(* Schneider Machine Expert - Basic project Temporizador, file version 2.7.0.0 *)
(* ProjectInformations: Name=Nuevo proyecto *)

HARDWARE
  Cpu 0: TM221C24R
  EthernetConfiguration: NetworkName=M221, IpAllocationMode=FixedAddress, IpAddress=0.0.0.0, SubnetMask=0.0.0.0
  SerialLineConfiguration: Baud=Baud19200, Parity=ParityEven, DataBits=DataBits8, StopBits=StopBits1, PhysicalMedium=PhysicalMediumRs485, TransmissionMode=TransmissionModeModbusRtu, SlaveId=1, Addressing=SlaveAddressing
  MastTask: UsePeriodScanMode=false, PeriodScan=100
  FastTask: Period=255
  CpuBehavior: StartingMode=StartAsPreviousState, AutoSaveRamOnEeprom=true, WatchdogPeriod=250

SYMBOLS  (address, symbol, comment, settings)
  %M0         "Fill"
  %M1         "Discharge"
  %M3         "Fill valve"
  %M4         "Fillin"
  %M5         "Discharge valve"
  %M6         "Discharging"
  %TM0        "Timer Fill"  [Type=TP, Preset=10, Base=OneSecond]
  %TM1        "Timer Discharge"  [Type=TP, Preset=10, Base=OneSecond]

POU Nuevo POU
  (* SectionNumber=1 *)

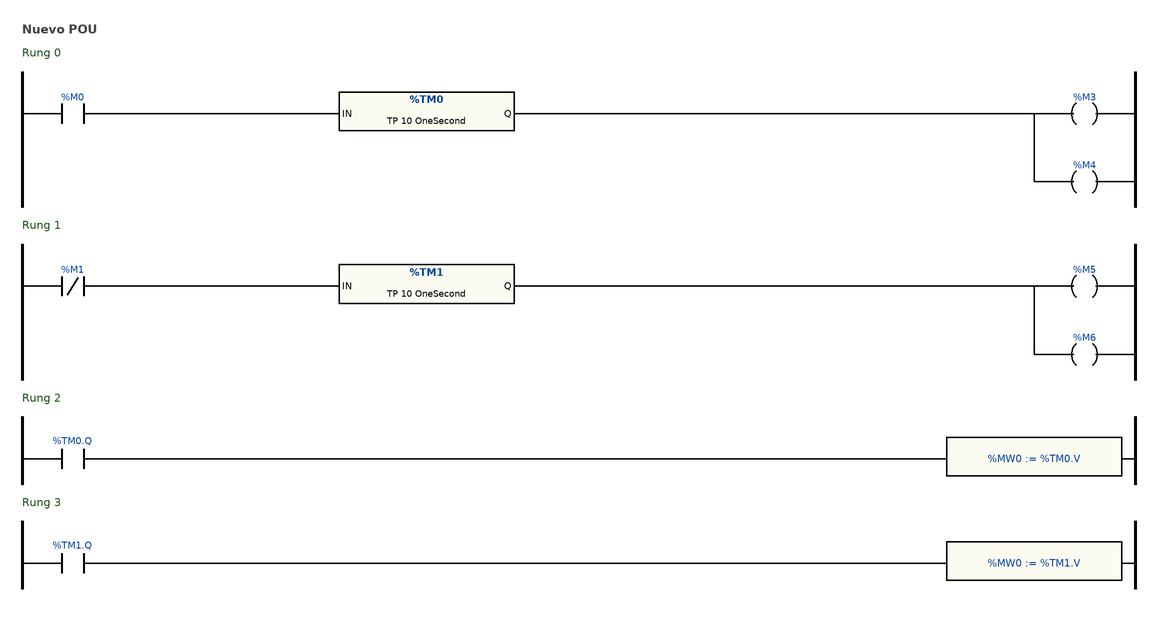

// Rung 0
  BLK %TM0
  LD %M0
  IN
  OUT_BLK
  LD Q
  ST %M3
  ST %M4
  END_BLK
  // as ST:
  //   %TM0(IN := %M0);
  //   %M3 := %TM0.Q;
  //   %M4 := %TM0.Q;

// Rung 1
  BLK %TM1
  LDN %M1
  IN
  OUT_BLK
  LD Q
  ST %M5
  ST %M6
  END_BLK
  // as ST:
  //   %TM1(IN := NOT %M1);
  //   %M5 := %TM1.Q;
  //   %M6 := %TM1.Q;

// Rung 2
  LD %TM0.Q
  [ %MW0 := %TM0.V ]
  // as ST:
  //   IF %TM0.Q THEN %MW0 := %TM0.V; END_IF;

// Rung 3
  LD %TM1.Q
  [ %MW0 := %TM1.V ]
  // as ST:
  //   IF %TM1.Q THEN %MW0 := %TM1.V; END_IF;
